// TIA Portal V18 export
ORGANIZATION_BLOCK "20-Autoleveler"   // OB133, LAD, ProgramCycle
TITLE = "Main Program Sweep (Cycle)"
{ S7_Optimized_Access := 'TRUE' }
VERSION : 0.1
// stored: AutoNumber true, IsIECCheckEnabled false, SetENOAutomatically false
   VAR_INPUT
      Initial_Call : Bool;   // Initial call of this OB
      Remanence : Bool;   // =True, if remanent data are available
   END_VAR
   VAR_TEMP   // added for the SCL form of the ladder/FBD networks
      _w1 : Bool;
      _w2 : Bool;
   END_VAR
BEGIN

REGION Network 1: AutoLeveller Definition
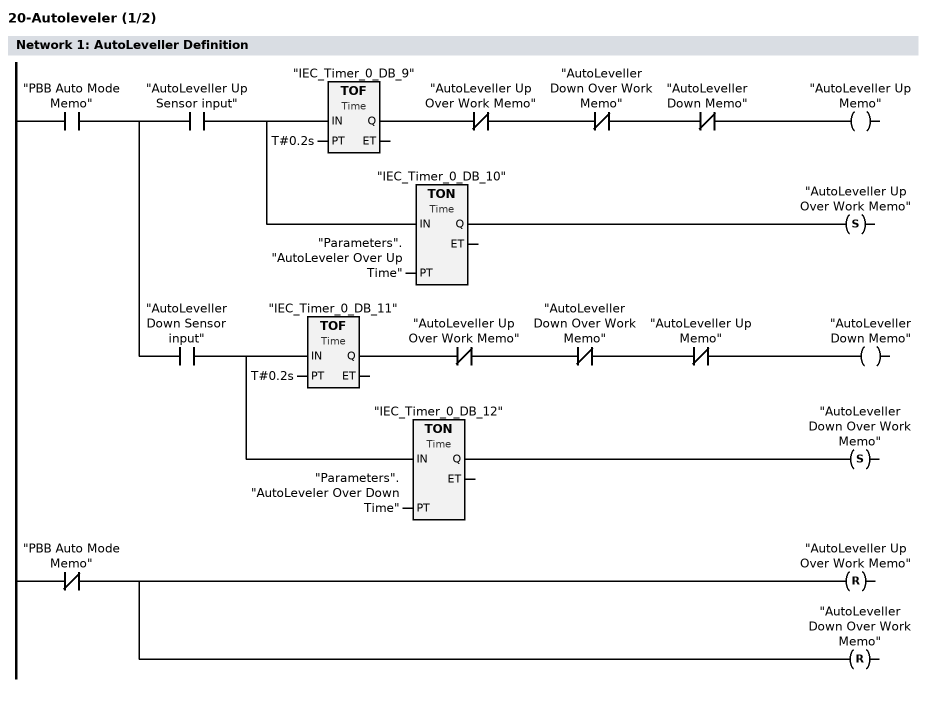
   RUNG wire#powerrail
      Contact( "PBB Auto Mode Memo" )
      wire#w1
      Contact( "AutoLeveller Up Sensor input" )
      wire#w2
      { S7_Templates := "time_type := Time" } "IEC_Timer_0_DB_9".TOF(pt := T#0.2s, et =>)
      I_Contact( "AutoLeveller Up Over Work Memo" )
      I_Contact( "AutoLeveller Down Over Work Memo" )
      I_Contact( "AutoLeveller Down Memo" )
      Coil( "AutoLeveller Up Memo" )
   END_RUNG
   RUNG wire#w2
      { S7_Templates := "time_type := Time" } "IEC_Timer_0_DB_10".TON(pt := "Parameters"."AutoLeveler Over Up Time", et =>)
      S_Coil( "AutoLeveller Up Over Work Memo" )
   END_RUNG
   RUNG wire#w1
      Contact( "AutoLeveller Down Sensor input" )
      wire#w3
      { S7_Templates := "time_type := Time" } "IEC_Timer_0_DB_11".TOF(pt := T#0.2s, et =>)
      I_Contact( "AutoLeveller Up Over Work Memo" )
      I_Contact( "AutoLeveller Down Over Work Memo" )
      I_Contact( "AutoLeveller Up Memo" )
      Coil( "AutoLeveller Down Memo" )
   END_RUNG
   RUNG wire#w3
      { S7_Templates := "time_type := Time" } "IEC_Timer_0_DB_12".TON(pt := "Parameters"."AutoLeveler Over Down Time", et =>)
      S_Coil( "AutoLeveller Down Over Work Memo" )
   END_RUNG
   RUNG wire#powerrail
      I_Contact( "PBB Auto Mode Memo" )
      wire#w4
      R_Coil( "AutoLeveller Up Over Work Memo" )
   END_RUNG
   RUNG wire#w4
      R_Coil( "AutoLeveller Down Over Work Memo" )
   END_RUNG
   // the same network as SCL:
   #_w1 := "PBB Auto Mode Memo" AND "AutoLeveller Up Sensor input";
   "IEC_Timer_0_DB_9".TOF(IN := #_w1, PT := T#0.2s);
   "AutoLeveller Up Memo" := "IEC_Timer_0_DB_9".Q AND NOT "AutoLeveller Up Over Work Memo" AND NOT "AutoLeveller Down Over Work Memo" AND NOT "AutoLeveller Down Memo";
   "IEC_Timer_0_DB_10".TON(IN := #_w1, PT := "Parameters"."AutoLeveler Over Up Time");
   IF "IEC_Timer_0_DB_10".Q THEN "AutoLeveller Up Over Work Memo" := TRUE; END_IF;
   #_w2 := "PBB Auto Mode Memo" AND "AutoLeveller Down Sensor input";
   "IEC_Timer_0_DB_11".TOF(IN := #_w2, PT := T#0.2s);
   "AutoLeveller Down Memo" := "IEC_Timer_0_DB_11".Q AND NOT "AutoLeveller Up Over Work Memo" AND NOT "AutoLeveller Down Over Work Memo" AND NOT "AutoLeveller Up Memo";
   "IEC_Timer_0_DB_12".TON(IN := #_w2, PT := "Parameters"."AutoLeveler Over Down Time");
   IF "IEC_Timer_0_DB_12".Q THEN "AutoLeveller Down Over Work Memo" := TRUE; END_IF;
   IF NOT "PBB Auto Mode Memo" THEN
       "AutoLeveller Up Over Work Memo" := FALSE;
       "AutoLeveller Down Over Work Memo" := FALSE;
   END_IF;
END_REGION

REGION Network 2: AutoLeveller Motor
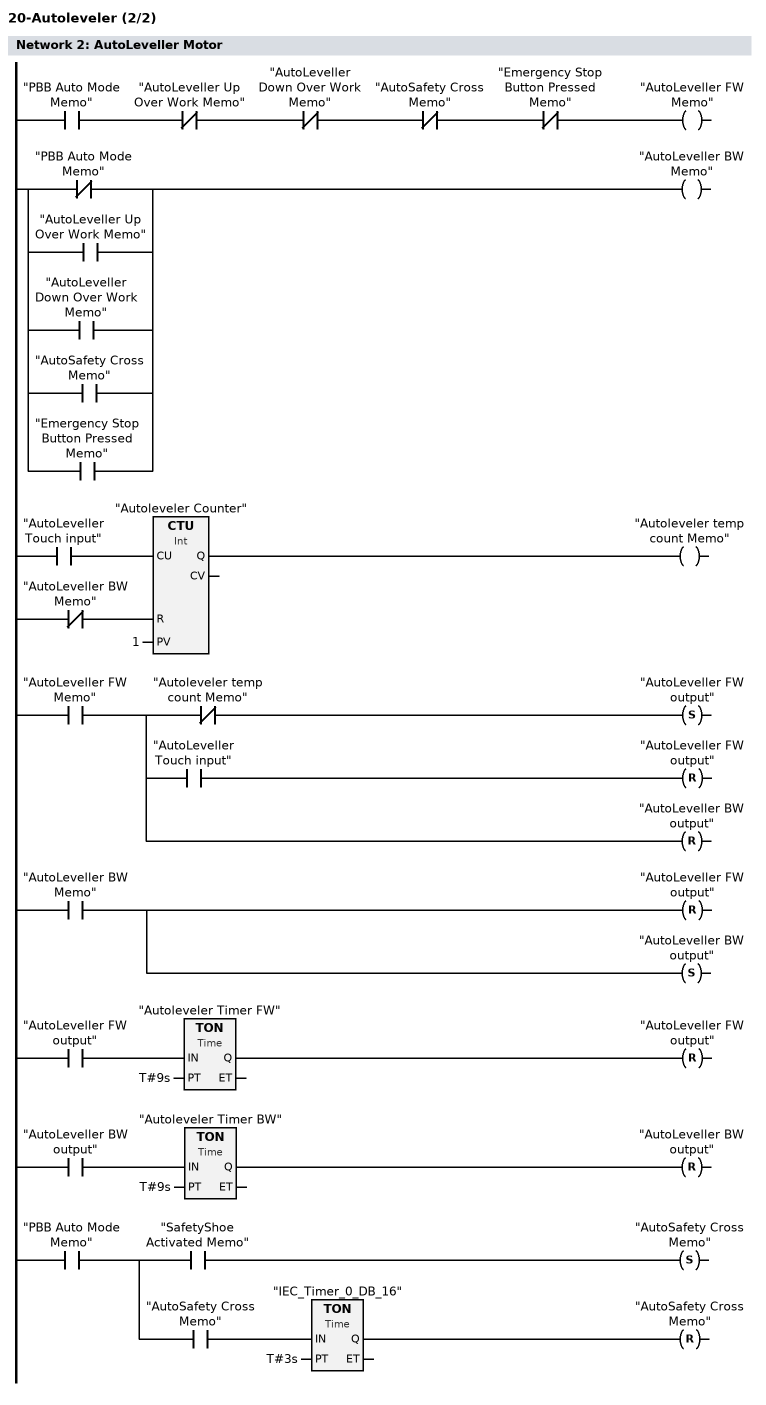
   RUNG wire#powerrail
      Contact( "PBB Auto Mode Memo" )
      I_Contact( "AutoLeveller Up Over Work Memo" )
      I_Contact( "AutoLeveller Down Over Work Memo" )
      I_Contact( "AutoSafety Cross Memo" )
      I_Contact( "Emergency Stop Button Pressed Memo" )
      Coil( "AutoLeveller FW Memo" )
   END_RUNG
   RUNG wire#powerrail
      I_Contact( "PBB Auto Mode Memo" )
      wire#w1
      Coil( "AutoLeveller BW Memo" )
   END_RUNG
   RUNG wire#powerrail
      Contact( "AutoLeveller Up Over Work Memo" )
   END_RUNG wire#w1
   RUNG wire#powerrail
      Contact( "AutoLeveller Down Over Work Memo" )
   END_RUNG wire#w1
   RUNG wire#powerrail
      Contact( "AutoSafety Cross Memo" )
   END_RUNG wire#w1
   RUNG wire#powerrail
      Contact( "Emergency Stop Button Pressed Memo" )
   END_RUNG wire#w1
   RUNG wire#powerrail
      Contact( "AutoLeveller Touch input" )
      { S7_Templates := "value_type := Int" } "Autoleveler Counter".CTU(r := wire#w2, pv := 1, cv =>)
      Coil( "Autoleveler temp count Memo" )
   END_RUNG
   RUNG wire#powerrail
      I_Contact( "AutoLeveller BW Memo" )
   END_RUNG wire#w2
   RUNG wire#powerrail
      Contact( "AutoLeveller FW Memo" )
      wire#w3
      I_Contact( "Autoleveler temp count Memo" )
      S_Coil( "AutoLeveller FW output" )
   END_RUNG
   RUNG wire#w3
      Contact( "AutoLeveller Touch input" )
      R_Coil( "AutoLeveller FW output" )
   END_RUNG
   RUNG wire#w3
      R_Coil( "AutoLeveller BW output" )
   END_RUNG
   RUNG wire#powerrail
      Contact( "AutoLeveller BW Memo" )
      wire#w4
      R_Coil( "AutoLeveller FW output" )
   END_RUNG
   RUNG wire#w4
      S_Coil( "AutoLeveller BW output" )
   END_RUNG
   RUNG wire#powerrail
      Contact( "AutoLeveller FW output" )
      { S7_Templates := "time_type := Time" } "Autoleveler Timer FW".TON(pt := T#9s, et =>)
      R_Coil( "AutoLeveller FW output" )
   END_RUNG
   RUNG wire#powerrail
      Contact( "AutoLeveller BW output" )
      { S7_Templates := "time_type := Time" } "Autoleveler Timer BW".TON(pt := T#9s, et =>)
      R_Coil( "AutoLeveller BW output" )
   END_RUNG
   RUNG wire#powerrail
      Contact( "PBB Auto Mode Memo" )
      wire#w5
      Contact( "SafetyShoe Activated Memo" )
      S_Coil( "AutoSafety Cross Memo" )
   END_RUNG
   RUNG wire#w5
      Contact( "AutoSafety Cross Memo" )
      { S7_Templates := "time_type := Time" } "IEC_Timer_0_DB_16".TON(pt := T#3s, et =>)
      R_Coil( "AutoSafety Cross Memo" )
   END_RUNG
   // the same network as SCL:
   "AutoLeveller FW Memo" := "PBB Auto Mode Memo" AND NOT "AutoLeveller Up Over Work Memo" AND NOT "AutoLeveller Down Over Work Memo" AND NOT "AutoSafety Cross Memo" AND NOT "Emergency Stop Button Pressed Memo";
   "AutoLeveller BW Memo" := NOT "PBB Auto Mode Memo" OR "AutoLeveller Up Over Work Memo" OR "AutoLeveller Down Over Work Memo" OR "AutoSafety Cross Memo" OR "Emergency Stop Button Pressed Memo";
   "Autoleveler Counter".CTU(CU := "AutoLeveller Touch input", R := NOT "AutoLeveller BW Memo", PV := 1);
   "Autoleveler temp count Memo" := "Autoleveler Counter".Q;
   IF "AutoLeveller FW Memo" AND NOT "Autoleveler temp count Memo" THEN
       "AutoLeveller FW output" := TRUE;
   END_IF;
   IF "AutoLeveller FW Memo" AND "AutoLeveller Touch input" THEN "AutoLeveller FW output" := FALSE; END_IF;
   IF "AutoLeveller FW Memo" THEN "AutoLeveller BW output" := FALSE; END_IF;
   IF "AutoLeveller BW Memo" THEN
       "AutoLeveller FW output" := FALSE;
       "AutoLeveller BW output" := TRUE;
   END_IF;
   "Autoleveler Timer FW".TON(IN := "AutoLeveller FW output", PT := T#9s);
   IF "Autoleveler Timer FW".Q THEN "AutoLeveller FW output" := FALSE; END_IF;
   "Autoleveler Timer BW".TON(IN := "AutoLeveller BW output", PT := T#9s);
   IF "Autoleveler Timer BW".Q THEN "AutoLeveller BW output" := FALSE; END_IF;
   IF "PBB Auto Mode Memo" AND "SafetyShoe Activated Memo" THEN "AutoSafety Cross Memo" := TRUE; END_IF;
   "IEC_Timer_0_DB_16".TON(IN := "PBB Auto Mode Memo" AND "AutoSafety Cross Memo", PT := T#3s);
   IF "IEC_Timer_0_DB_16".Q THEN "AutoSafety Cross Memo" := FALSE; END_IF;
END_REGION
END_ORGANIZATION_BLOCK
